PROGRAM MAIN
VAR
	{attribute 'pytmc' := 'pv: PREFIX:fbTest'}
	fbTest : FB_SampleA_Test;
	{attribute 'pytmc' := 'pv: PREFIX:fOutput'}
	fOutput : LREAL;
END_VAR

fbTest(fInput:=1.0, fOutput=>fOutput);

END_PROGRAM

(* stored: Version 1.1.0.1, ProductVersion 3.1.4022.18
   POU MAIN: Id {84dff641-e6f4-4dbd-8059-d7804ecb70ca}, SpecialFunc None *)
